FUNCTION_BLOCK EquipmentModule EXTENDS FB_PackML_BaseModule IMPLEMENTS ITF_Observer
VAR
	//data from Observable
	data : UDINT;
END_VAR

METHOD PUBLIC CyclicLogic
VAR
	i : UDINT;
END_VAR
IF NOT _InitComplete THEN
	_InitComplete := Initialize();
	RETURN;
END_IF
END_METHOD

METHOD PROTECTED Initialize : BOOL
Initialize := true;
END_METHOD

METHOD update : BOOL
VAR_INPUT
	Module : REFERENCE TO MachineModule;
END_VAR
//Get desired info from Observable
data := Module.Data;
END_METHOD

END_FUNCTION_BLOCK

(* stored: Version 1.1.0.1, ProductVersion 3.1.4024.12
   POU EquipmentModule: Id {c012c6f7-cfaf-489a-882b-e9bef571a81f}, SpecialFunc None
   Method CyclicLogic: Id {97e9fea4-c26f-4ae1-830e-87fb3563d9c6}
   Method Initialize: Id {507e7079-319d-4c87-9253-ef7b1ad19c7f}
   Method update: Id {1ff49e6f-cd52-4f76-b086-59f66795e98d} *)
